// Mitsubishi GX Works2 project: timer1   PLC: Q03UDV

PROGRAM MAIN
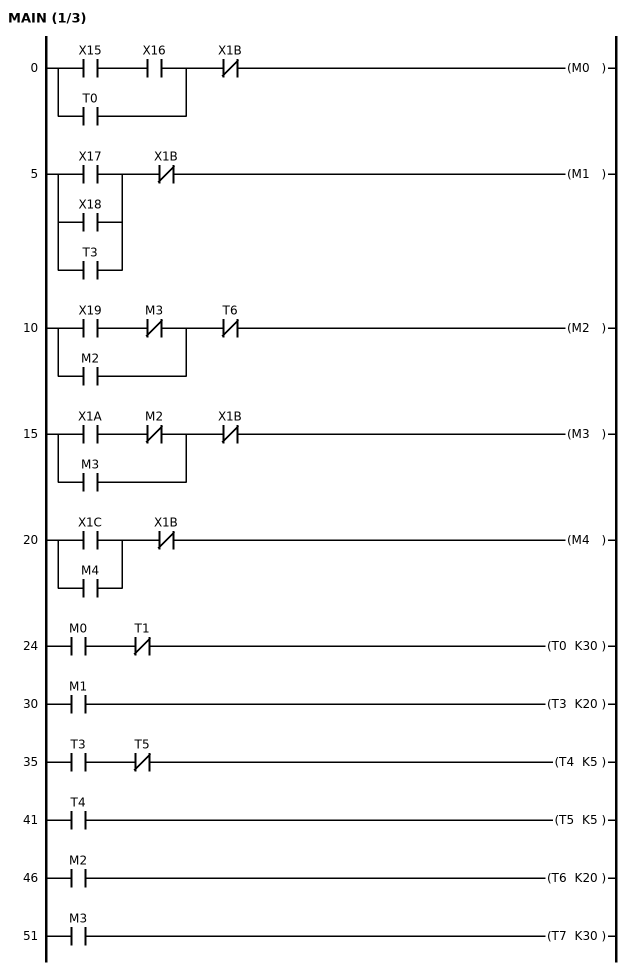
0     LD      X15
      AND     X16
      OR      T0
      ANI     X1B
      OUT     M0
5     LD      X17
      OR      X18
      OR      T3
      ANI     X1B
      OUT     M1
10    LD      X19
      ANI     M3
      OR      M2
      ANI     T6
      OUT     M2
15    LD      X1A
      ANI     M2
      OR      M3
      ANI     X1B
      OUT     M3
20    LD      X1C
      OR      M4
      ANI     X1B
      OUT     M4
24    LD      M0
      ANI     T1
      OUT     T0 K30
30    LD      M1
      OUT     T3 K20
35    LD      T3
      ANI     T5
      OUT     T4 K5
41    LD      T4
      OUT     T5 K5
46    LD      M2
      OUT     T6 K20
51    LD      M3
      OUT     T7 K30
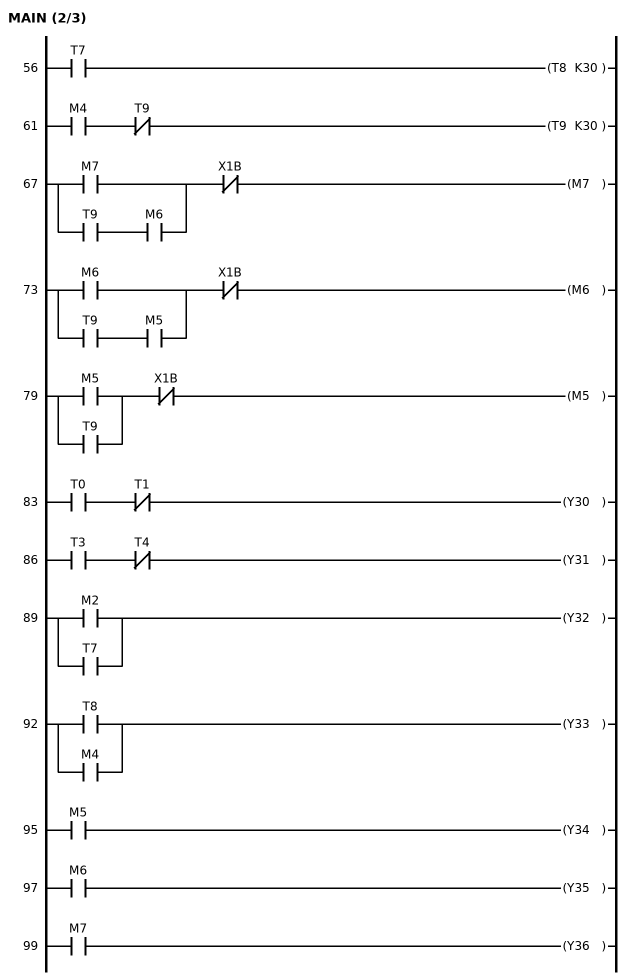
56    LD      T7
      OUT     T8 K30
61    LD      M4
      ANI     T9
      OUT     T9 K30
67    LD      M7
      LD      T9
      AND     M6
      ORB
      ANI     X1B
      OUT     M7
73    LD      M6
      LD      T9
      AND     M5
      ORB
      ANI     X1B
      OUT     M6
79    LD      M5
      OR      T9
      ANI     X1B
      OUT     M5
83    LD      T0
      ANI     T1
      OUT     Y30
86    LD      T3
      ANI     T4
      OUT     Y31
89    LD      M2
      OR      T7
      OUT     Y32
92    LD      T8
      OR      M4
      OUT     Y33
95    LD      M5
      OUT     Y34
97    LD      M6
      OUT     Y35
99    LD      M7
      OUT     Y36
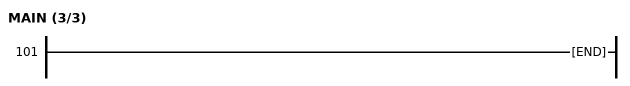
101   END
END_PROGRAM
